Staubli VAL3: Form_Action.pgx

public program Form_Action(string x_sTitle, string x_sPanelTitle, string& x_sList[], num& x_nSelectIndex, bool& x_bIO[], num x_nPresetIndex, string& x_sLable[])
  local num l_nNum
begin
  //为lasman3.0进行配置界面
 // cls()
  x_nSelectIndex=round(x_nSelectIndex)%500
  x_nPresetIndex=x_nPresetIndex%50
  title(x_sTitle)
   gotoxy(0,0)
  put("动作执行需上电!")
  gotoxy(0,2)
  put("动作参数:")





  call Control_PanelXY(22,0,15,10)
    for l_nNum=0 to size(x_sLable)-1
    gotoxy(0,l_nNum+3)
    put(left(x_sLable[l_nNum]+"                            ",nPanelLTopX-1))
    endFor
  call Control_Panel(x_sPanelTitle)
  setTextMode(sel(x_bIO[0],1,0))
  gotoxy(1,13)
  put("执行")

 setTextMode(0)

        gotoxy(21,13)
    put("上传")
    gotoxy(31,13)
    put("保存")

    gotoxy(26,13)
    put("修改")
    gotoxy(31,13)
    put("保存")

    gotoxy(36,13)
    put("退出")


  call Control_List(x_sList,x_nSelectIndex)



end
